// TIA Portal V20 export
TYPE "LWONIK_typeDoorControlNodes"
// stored: Access Published
   STRUCT
      commands : Struct
         Front_UnwinderDoorSelect : Bool;
         Front_NotchingDoorSelect : Bool;
         Front_VisionDoorSelect : Bool;
         Rear_UnwinderDoorSelect : Bool;
         Rear_NotchingDoorSelect : Bool;
         Rear_VisionDoorSelect : Bool;
         Rear_RewinderDoorSelect : Bool;
         Rear_ScrapCutterDoorSelect : Bool;
         DoorLock : Bool;
         DoorUnlock : Bool;
      END_STRUCT;
      monitoring : Struct
         Front_UnwinderDoorSelect : Bool;
         Front_NotchingDoorSelect : Bool;
         Front_VisionDoorSelect : Bool;
         Rear_UnwinderDoorSelect : Bool;
         Rear_NotchingDoorSelect : Bool;
         Rear_VisionDoorSelect : Bool;
         Rear_RewinderDoorSelect : Bool;
         Rear_ScrapCutterDoorSelect : Bool;
         DoorLock : Bool;
         DoorUnlock : Bool;
      END_STRUCT;
   END_STRUCT;
END_TYPE
